{attribute 'linkalways'} 
{attribute 'no_explicit_call' := 'This FB is a CLASS and must be accessed using methods or properties'}
{attribute 'enable_dynamic_creation'}
FUNCTION_BLOCK Node_F_VN_DeinitializeFunction EXTENDS VisionNode
VAR
    eFunction : _ETcVnInitializableFunction(ETcVnInitializableFunction.TCVN_IF_OCR);
    nOptions : _ULINT(0);
    hrPrev : _HRESULT(S_OK);
	hresult : _HRESULT(S_OK);
END_VAR

METHOD PUBLIC  Clone : I_Node
VAR
	pNode : POINTER TO Node_F_VN_DeinitializeFunction;
END_VAR
pNode := __NEW(Node_F_VN_DeinitializeFunction);
Clone := pNode^;
END_METHOD

METHOD FB_init : BOOL
VAR_INPUT
	bInitRetains : BOOL; // if TRUE, the retain variables are initialized (warm start / cold start)
	bInCopyCode : BOOL;  // if TRUE, the instance afterwards gets moved into the copy code (online change)
END_VAR
AddParameter('eFunction', eFunction);
AddParameter('nOptions', nOptions);
AddInput('hrPrev', hrPrev);
AddOutput('hresult',hresult);
END_METHOD

METHOD PROTECTED OnExecute
hresult.Value := F_VN_DeinitializeFunction(
	eFunction := eFunction.Value,
    nOptions := nOptions.Value,
	hrPrev:= hrPrev.Value);
END_METHOD

METHOD PUBLIC PreExecutionCheck
VAR_INPUT
	Check : I_PreExecutionChecks;
END_VAR
END_METHOD

END_FUNCTION_BLOCK

(* stored: Version 1.1.0.1, ProductVersion 3.1.4024.13
   POU Node_F_VN_DeinitializeFunction: Id {61b0422a-8aaa-083a-083c-30c63c098b81}, SpecialFunc None
   Folder Constructor: Id {8aae284b-97a0-084a-0190-6f6283c55ebb}
   Method Clone: Id {bcedb33c-210b-0e0a-3b1a-0b9a394368e9}
   Method FB_init: Id {f16b0e5f-e89e-0536-2271-8c2b48308a06}
   Method OnExecute: Id {c169e431-a005-0ce9-0d01-b739e364531a}
   Method PreExecutionCheck: Id {593449b3-3243-0c29-32ff-ec559cb9da1a} *)
